{attribute 'qualified_only'}
{attribute 'strict'}
TYPE eP_direction :
(
	keep :=0,
	negative,
	positive
);
END_TYPE

(* stored: Version 1.1.0.1, ProductVersion 3.1.4024.11
   DUT eP_direction: Id {9c60b105-6cdd-4450-bd7b-2d96953a808e} *)
